# EPICS StreamDevice protocol: proto/pfeiffer.proto
Terminator = CR;

writePumpOn {
	out "\$11001206000000%+<sum>";
	in  "\$11001206000000%+<sum>";
	out "\$11001006111111%+<sum>";
	in  "\$11001006111111%+<sum>";
}

writePumpOff {
	out "\$11001206000000%+<sum>";
	in  "\$11001206000000%+<sum>";
	out "\$11001006000000%+<sum>";
	in  "\$11001006000000%+<sum>";
}

writePumpOffVent {
	out "\$11001206111111%+<sum>";
	in  "\$11001206111111%+<sum>";
	out "\$11001006000000%+<sum>";
	in  "\$11001006000000%+<sum>";
}

readBoolParam {
	out "\$100\$202=?%+<sum>";
	in "\$110\$206%{000000|111111}%+<sum>";
}

writeBoolParam {
	out "\$110\$206%{000000|111111}%+<sum>";
	in "\$110\$206%{000000|111111}%+<sum>";
}

readIntParam {
	out "\$100\$202=?%+<sum>";
	in "\$110\$206%6d%+<sum>";
}

writeIntParam {
	out "\$110\$206%06d%+<sum>";
	in "\$110\$206%6d%+<sum>";
}

readShortIntParam {
	out "\$100\$202=?%+<sum>";
	in "\$110\$203%3d%+<sum>";
}

writeShortIntParam {
	out "\$110\$203%03d%+<sum>";
	in "\$110\$203%3d%+<sum>";
}

readStringParam {
	out "\$100\$202=?%+<sum>";
	in "\$110\$206%6s%+<sum>";
}

writeStringParam {
	out "\$100\$206%6s%+<sum>";
	in "\$110\$206%6s%+<sum>";
}

readErrorParam {
	out "\$100\$202=?%+<sum>";
	in "\$110\$206%{000|Wrn|Err}%*3d%+<sum>";
}

readErrorCodeParam {
	out "\$100\$202=?%+<sum>";
	in "\$110\$206%*{000|Wrn|Err}%3d%+<sum>";
}
